FUNCTION_BLOCK BaseGripper
VAR_INPUT
END_VAR
VAR_OUTPUT
END_VAR
VAR
END_VAR

END_FUNCTION_BLOCK

(* stored: Version 1.1.0.1
   POU BaseGripper: Id {328c9d79-6f6a-4f42-95c9-9fd65dfe9285}, SpecialFunc None *)
